FUNCTION BreedCalculation
VAR_INPUT
END_VAR
VAR
	sizeMeasure : SizeMeasure;
	weightMeasure : WeightMeasure;
END_VAR

sizeMeasure();
weightMeasure();
//Insted of a new object, just call the global object from the main
//MAIN.sizeMeasure.sizeInCm;

//Small and non metal. Bin1 breed
IF (sizeMeasure.sizeInCm >= 10.0 AND sizeMeasure.sizeInCm <= 20.0 AND weightMeasure.weightInKg <= 5.0 AND
	NOT MeasuringData.MetalMaterial) THEN
	MeasuringData.Bin1Breed := TRUE;
	MeasuringData.Bin2Breed := FALSE;
	MeasuringData.Bin3Breed := FALSE;
	MeasuringData.Bin4Breed := FALSE;
END_IF

//Small and metal. Bin2 breed
IF (sizeMeasure.sizeInCm >= 10.0 AND sizeMeasure.sizeInCm <= 20.0 AND weightMeasure.weightInKg <= 5.0 AND
	MeasuringData.MetalMaterial) THEN
	MeasuringData.Bin1Breed := FALSE;
	MeasuringData.Bin2Breed := TRUE;
	MeasuringData.Bin3Breed := FALSE;
	MeasuringData.Bin4Breed := FALSE;
END_IF

//Large and non metal. Bin3 breed
IF (sizeMeasure.sizeInCm >= 20.0 AND weightMeasure.weightInKg >= 5.1 AND
	NOT MeasuringData.MetalMaterial) THEN
	MeasuringData.Bin1Breed := FALSE;
	MeasuringData.Bin2Breed := FALSE;
	MeasuringData.Bin3Breed := TRUE;
	MeasuringData.Bin4Breed := FALSE;
END_IF

//Large and metal. Bin4 breed
IF (sizeMeasure.sizeInCm >= 20.0 AND weightMeasure.weightInKg >= 5.1 AND
	MeasuringData.MetalMaterial) THEN
	MeasuringData.Bin1Breed := FALSE;
	MeasuringData.Bin2Breed := FALSE;
	MeasuringData.Bin3Breed := FALSE;
	MeasuringData.Bin4Breed := TRUE;
END_IF

END_FUNCTION

(* stored: Version 1.1.0.1, ProductVersion 3.1.4024.13
   POU BreedCalculation: Id {a45dfa7e-50d0-46f2-8d49-26b35c643089}, SpecialFunc None *)
